(* CoDeSys 2.3 export: NETVAROD_UDP.EXP *)

(* Data type *)
TYPE NetVarOD_UDP :
STRUCT
	(* Variablen, die bei der Initialaisierung übergeben werden *)
	pPtr				: POINTER TO ARRAY[0..255] OF BYTE;
	nIndex				: INT;
	nSubIndex			: INT;
	nItems				: INT;
	nItemLen			: INT;
	byAccess			: BYTE;
	byAttrib			: BYTE;
END_STRUCT
END_TYPE
